% RSLogix 500 project Q13.RSS, saved by version 8.30.00.16 %
PROJECT "Q13"    % processor: Bul.1763 MicroLogix 1100 Series B %

PROGRAM FILES
  LAD 2   7 rungs

DATA FILES
  O0 OUTPUT  4 elements
  I1 INPUT  6 elements
  S2 STATUS  66 elements
  B3 BINARY  1 elements
  T4 TIMER  1 elements
  C5 COUNTER  1 elements
  R6 CONTROL  1 elements
  N7 INTEGER  1 elements
  F8 FLOAT  1 elements

LADDER 2
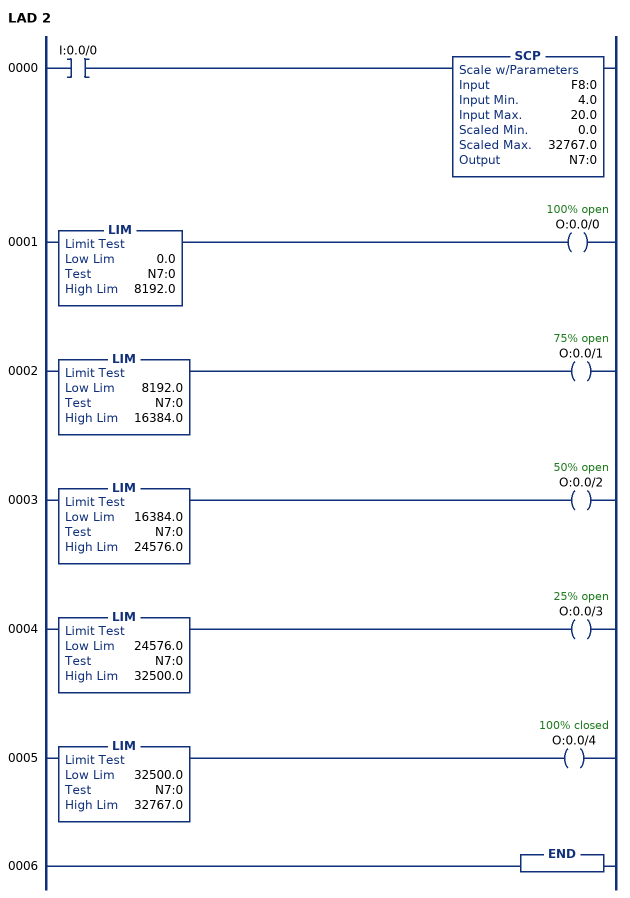
% Rung: 0 %
SOR XIC I:0.0/0 SCP F8:0 4.0 20.0 0.0 32767.0 N7:0 EOR
% Rung: 1 %
SOR LIM 0.0 N7:0 8192.0 OTE O:0.0/0 EOR
%   O:0.0/0  "100% open" %
% Rung: 2 %
SOR LIM 8192.0 N7:0 16384.0 OTE O:0.0/1 EOR
%   O:0.0/1  "75% open" %
% Rung: 3 %
SOR LIM 16384.0 N7:0 24576.0 OTE O:0.0/2 EOR
%   O:0.0/2  "50% open" %
% Rung: 4 %
SOR LIM 24576.0 N7:0 32500.0 OTE O:0.0/3 EOR
%   O:0.0/3  "25% open" %
% Rung: 5 %
SOR LIM 32500.0 N7:0 32767.0 OTE O:0.0/4 EOR
%   O:0.0/4  "100% closed" %
% Rung: 6 %
SOR END EOR

DATA TABLE (non-zero values as saved)
DATA F8
% F8:0 % 6
